FUNCTION_BLOCK SafetyHydraulicsAndSafetyIO EXTENDS SM_SafetyHydraulicsAndSafetyIO
VAR_INPUT
END_VAR
VAR_OUTPUT
END_VAR
VAR
    _testVar : INT;
END_VAR

SUPER^();

// do stuff

//SUPER^();

END_FUNCTION_BLOCK

(* stored: Version 1.1.0.1, ProductVersion 3.1.4018.5
   POU SafetyHydraulicsAndSafetyIO: Id {fafd51c0-7c66-4aff-89a1-c11a6e3c5ddf}, SpecialFunc None *)
